TYPE "udtRackAI"
VERSION : 0.1
   STRUCT
      IW_ReservoirLevel { ExternalAccessible := 'False'; ExternalVisible := 'False'; ExternalWritable := 'False'} : Int;
   END_STRUCT;

END_TYPE

